TYPE ST_TxUdpRemote :
STRUCT
	t : REAL;
	em8000 : ST_FeedbackStewart;
	em1500 : ST_FeedbackStewart;
	comau : ST_FeedbackComau;
	at960 : ST_FeedbackLeica;
	mru1 : ST_FeedbackMru;
	mru2 : ST_FeedbackMru;
	markers : ARRAY [0..9] OF ST_3DMarkerPositionNoLabel;
	winch : ST_FeedbackWinch;
END_STRUCT
END_TYPE

(* stored: Version 1.1.0.1, ProductVersion 3.1.4022.7
   DUT ST_TxUdpRemote: Id {e855cfb6-bd67-4fa5-9051-ffcbcaa8ada0} *)
